// Operator action journal
IF GVL_STATUS.G_Diagnostics.Operator_Action_Blocked AND NOT L_Last_Operator_Blocked THEN
    GVL_STATUS.G_Diagnostics.Operator_Journal_Event_Seq := GVL_STATUS.G_Diagnostics.Operator_Journal_Event_Seq + 1;
END_IF;
L_Last_Operator_Blocked := GVL_STATUS.G_Diagnostics.Operator_Action_Blocked;
IF GVL_CONFIG.G_DHW_Heating_Pump_In_Service <> L_Last_DHW_Heating_In_Service THEN
    GVL_STATUS.G_Diagnostics.Operator_Journal_Event_Seq := GVL_STATUS.G_Diagnostics.Operator_Journal_Event_Seq + 1;
    IF GVL_CONFIG.G_DHW_Heating_Pump_In_Service THEN
        GVL_STATUS.G_Diagnostics.Maintenance_Last_Action := 'Насос загрузки ГВС возвращён из ТО';
    ELSE
        GVL_STATUS.G_Diagnostics.Maintenance_Last_Action := 'Насос загрузки ГВС выведен в ТО';
    END_IF;
END_IF;
L_Last_DHW_Heating_In_Service := GVL_CONFIG.G_DHW_Heating_Pump_In_Service;
IF GVL_CONFIG.G_DHW_Circ_Pump_In_Service <> L_Last_DHW_Circ_In_Service THEN
    GVL_STATUS.G_Diagnostics.Operator_Journal_Event_Seq := GVL_STATUS.G_Diagnostics.Operator_Journal_Event_Seq + 1;
    IF GVL_CONFIG.G_DHW_Circ_Pump_In_Service THEN
        GVL_STATUS.G_Diagnostics.Maintenance_Last_Action := 'Насос рециркуляции ГВС возвращён из ТО';
    ELSE
        GVL_STATUS.G_Diagnostics.Maintenance_Last_Action := 'Насос рециркуляции ГВС выведен в ТО';
    END_IF;
END_IF;
L_Last_DHW_Circ_In_Service := GVL_CONFIG.G_DHW_Circ_Pump_In_Service;
IF GVL_STATUS.G_Diagnostics.Operator_Journal_Event_Seq <> GVL_STATUS.G_Diagnostics.Operator_Journal_Last_Seq THEN
    GVL_STATUS.G_Diagnostics.Operator_Journal_3 := GVL_STATUS.G_Diagnostics.Operator_Journal_2;
    GVL_STATUS.G_Diagnostics.Operator_Journal_2 := GVL_STATUS.G_Diagnostics.Operator_Journal_1;
    IF GVL_STATUS.G_Diagnostics.Operator_Last_Forbidden_Action <> '' THEN
        GVL_STATUS.G_Diagnostics.Operator_Journal_1 := GVL_STATUS.G_Diagnostics.Operator_Last_Forbidden_Action;
    ELSE
        GVL_STATUS.G_Diagnostics.Operator_Journal_1 := GVL_STATUS.G_Diagnostics.Maintenance_Last_Action;
    END_IF;
    GVL_STATUS.G_Diagnostics.Operator_Journal_Last_Seq := GVL_STATUS.G_Diagnostics.Operator_Journal_Event_Seq;
END_IF;

// ========================================
// CoreKernel live observer (diagnostic only)
// ========================================
// fbCoreKernelObserver disabled temporarily


// === NVRAM SNAPSHOT VIA STRUCT ADAPTER ===
L_Persist_Struct.System_Mode := GVL_STATE.G_System_Mode;

L_Persist_Struct.Safety_Gas_Latched := GVL_STATE.G_Safety_Gas_Latched;
L_Persist_Struct.Safety_Smoke_Latched := GVL_STATE.G_Safety_Smoke_Latched;
L_Persist_Struct.Safety_Leak_Latched := GVL_STATE.G_Safety_Leak_Latched;

L_Persist_Struct.DHW_Heating_Pump := GVL_STATE.G_DHW_Heating_Pump;
L_Persist_Struct.Valid := TRUE;

// mirror to legacy persistent variables
GVL_PERSISTENT.P_System_Mode := L_Persist_Struct.System_Mode;

GVL_PERSISTENT.P_Safety_Gas_Latched := L_Persist_Struct.Safety_Gas_Latched;
GVL_PERSISTENT.P_Safety_Smoke_Latched := L_Persist_Struct.Safety_Smoke_Latched;
GVL_PERSISTENT.P_Safety_Leak_Latched := L_Persist_Struct.Safety_Leak_Latched;

GVL_PERSISTENT.P_DHW_Heating_Active := L_Persist_Struct.DHW_Heating_Pump;
GVL_PERSISTENT.P_Valid := L_Persist_Struct.Valid;

// >>> BULK_SYNC_ANCHOR: PRG_System <<<

// === EVENT LOGGING: SCENARIO CHANGE ===
IF L_Scenario_Changed THEN
    fbLogEvent(
        VI_Event_Type := 1,
        VI_Timestamp := GVL_STATUS.G_System_Time_MS,
        VI_Param1 := TO_UDINT(L_Scenario_Source),
        VI_Param2 := TO_UDINT(L_Scenario_Intent)
    );
END_IF;

// === EVENT LOGGING: FAULTS ===

// IO
IF GVL_STATUS.G_Diagnostics.IO_Offline AND NOT L_IO_Fault_Prev THEN
    fbLogEvent(
        VI_Event_Type := 2,
        VI_Timestamp := GVL_STATUS.G_System_Time_MS,
        VI_Param1 := 1,
        VI_Param2 := 1
    );
END_IF;

IF NOT GVL_STATUS.G_Diagnostics.IO_Offline AND L_IO_Fault_Prev THEN
    fbLogEvent(
        VI_Event_Type := 3,
        VI_Timestamp := GVL_STATUS.G_System_Time_MS,
        VI_Param1 := 1,
        VI_Param2 := 0
    );
END_IF;

L_IO_Fault_Prev := GVL_STATUS.G_Diagnostics.IO_Offline;

// === EVENT LOGGING: MODE CHANGE ===
IF GVL_STATE.G_System_Mode <> L_Mode_Prev THEN
    fbLogEvent(
        VI_Event_Type := 4,
        VI_Timestamp := GVL_STATUS.G_System_Time_MS,
        VI_Param1 := TO_UDINT(L_Mode_Prev),
        VI_Param2 := TO_UDINT(GVL_STATE.G_System_Mode)
    );
END_IF;

L_Mode_Prev := GVL_STATE.G_System_Mode;
          
END_PROGRAM

PROGRAM PRG_System_Test_Harness
  VAR
    L_i : INT;
    L_j : INT;
    L_Used : REAL;
    L_HP_Used : REAL;
    L_HP_Manifold_Adjusted : ARRAY[1..GVL_CONSTANTS.C_MAX_MANIFOLDS] OF INT;
    fbDecisionTest : FB_Heating_Decision_Context;
    fbDecisionHP : FB_Heating_Decision_Context;
    fbTestResult : FB_Test_Result_Handler;
    fbTrace : FB_Trace_Logger;
  END_VAR

            IF NOT GVL_TEST.G_Test_Enable THEN
    RETURN;
END_IF;

GVL_TEST.G_Test_Total_Checks := 0;
GVL_TEST.G_Test_Failed_Checks := 0;
GVL_TEST.G_Test_Passed := TRUE;
GVL_TEST.G_Test_Last_Failure_Index := 0;
GVL_TEST.G_Test_Last_Failure_Code := 0;

// Reset transient failure flags for this scan
GVL_TEST.G_Diagnostics_Duplicate_Event_Found := FALSE;
GVL_TEST.G_Diagnostics_Count_Out_Of_Range := FALSE;
GVL_TEST.G_Heating_Allocation_Budget_Exceeded := FALSE;
GVL_TEST.G_Heating_Allocation_Enabled_Not_Allowed := FALSE;
GVL_TEST.G_Safety_Latched_Without_Intent := FALSE;
GVL_TEST.G_HP_Adjusted_Priority_Lower_Bound_Violation := FALSE;
GVL_TEST.G_HP_Adjusted_Allocation_Budget_Exceeded := FALSE;
GVL_TEST.G_HP_Adjusted_Allocation_Enabled_Not_Allowed := FALSE;
GVL_TEST.G_HP_Guest_Preheat_Config_Out_Of_Range := FALSE;

// =========================
// TEST 1: Diagnostics count bounds
// =========================
GVL_TEST.G_Test_Total_Checks := GVL_TEST.G_Test_Total_Checks + 1;
IF (GVL_STATUS.G_Diagnostics_Count < 0) OR (GVL_STATUS.G_Diagnostics_Count > 50) THEN
    GVL_TEST.G_Diagnostics_Count_Out_Of_Range := TRUE;
    GVL_TEST.G_Test_Failed_Checks := GVL_TEST.G_Test_Failed_Checks + 1;
    GVL_TEST.G_Test_Passed := FALSE;
    GVL_TEST.G_Test_Last_Failure_Index := 1;
    GVL_TEST.G_Test_Last_Failure_Code := 1001;
END_IF;

// =========================
// TEST 2: Diagnostics duplicates
// =========================
GVL_TEST.G_Test_Total_Checks := GVL_TEST.G_Test_Total_Checks + 1;
FOR L_i := 1 TO GVL_STATUS.G_Diagnostics_Count DO
    FOR L_j := L_i + 1 TO GVL_STATUS.G_Diagnostics_Count DO
        IF (GVL_STATUS.G_Diagnostics_Events[L_i].Code = GVL_STATUS.G_Diagnostics_Events[L_j].Code) AND
           (GVL_STATUS.G_Diagnostics_Events[L_i].Source = GVL_STATUS.G_Diagnostics_Events[L_j].Source) THEN
            GVL_TEST.G_Diagnostics_Duplicate_Event_Found := TRUE;
            GVL_TEST.G_Test_Failed_Checks := GVL_TEST.G_Test_Failed_Checks + 1;
            GVL_TEST.G_Test_Passed := FALSE;
            GVL_TEST.G_Test_Last_Failure_Index := 2;
            GVL_TEST.G_Test_Last_Failure_Code := 1002;
        END_IF;
    END_FOR;
END_FOR;

// =========================
// TEST 3: Base heating decision consistency
// =========================
GVL_TEST.G_Test_Total_Checks := GVL_TEST.G_Test_Total_Checks + 1;
fbDecisionTest(
    VI_Manifold_Pump_In_Service := GVL_CONFIG.G_Manifold_Pump_In_Service,
    VI_Manifold_Pressure_Fault := GVL_STATUS.G_Diagnostics.Manifold_Pressure_Fault,
    VI_Manifold_Current_Fault := GVL_STATUS.G_Diagnostics.Manifold_Current_Fault,
    VI_Manifold_Thermal_Weight := GVL_CONFIG.G_Manifold_Thermal_Weight,
    VI_Manifold_Priority := GVL_CONFIG.G_Manifold_Priority,
    VI_Max_Thermal_Budget := GVL_CONFIG.G_Max_Thermal_Budget
);

L_Used := 0.0;
FOR L_i := 1 TO GVL_CONSTANTS.C_MAX_MANIFOLDS DO
    IF fbDecisionTest.VO_Manifold_Enabled[L_i] AND (NOT fbDecisionTest.VO_Manifold_Allowed[L_i]) THEN
        GVL_TEST.G_Heating_Allocation_Enabled_Not_Allowed := TRUE;
        GVL_TEST.G_Test_Failed_Checks := GVL_TEST.G_Test_Failed_Checks + 1;
        GVL_TEST.G_Test_Passed := FALSE;
        GVL_TEST.G_Test_Last_Failure_Index := 3;
        GVL_TEST.G_Test_Last_Failure_Code := 1003;
    END_IF;

    IF fbDecisionTest.VO_Manifold_Enabled[L_i] THEN
        L_Used := L_Used + GVL_CONFIG.G_Manifold_Thermal_Weight[L_i];
    END_IF;
END_FOR;

IF L_Used > (GVL_CONFIG.G_Max_Thermal_Budget + 0.001) THEN
    GVL_TEST.G_Heating_Allocation_Budget_Exceeded := TRUE;
    GVL_TEST.G_Test_Failed_Checks := GVL_TEST.G_Test_Failed_Checks + 1;
    GVL_TEST.G_Test_Passed := FALSE;
    GVL_TEST.G_Test_Last_Failure_Index := 3;
    GVL_TEST.G_Test_Last_Failure_Code := 1004;
END_IF;

// =========================
// TEST 4: Safety latch consistency
// =========================
GVL_TEST.G_Test_Total_Checks := GVL_TEST.G_Test_Total_Checks + 1;
IF GVL_STATE.G_Safety_Gas_Latched AND (NOT GVL_INTENT_SAFETY.I_Gas_Alarm_Active) THEN
    GVL_TEST.G_Safety_Latched_Without_Intent := TRUE;
    GVL_TEST.G_Test_Failed_Checks := GVL_TEST.G_Test_Failed_Checks + 1;
    GVL_TEST.G_Test_Passed := FALSE;
    GVL_TEST.G_Test_Last_Failure_Index := 4;
    GVL_TEST.G_Test_Last_Failure_Code := 1005;
END_IF;

// =========================
// TEST 5: HP policy adjusted priority
// =========================
GVL_TEST.G_Test_Total_Checks := GVL_TEST.G_Test_Total_Checks + 1;

IF (GVL_HEATING_POLICY_CONFIG.G_Guest_Preheat_Priority_Boost < 0) OR (GVL_HEATING_POLICY_CONFIG.G_Guest_Preheat_Priority_Boost > 10) THEN
    GVL_TEST.G_HP_Guest_Preheat_Config_Out_Of_Range := TRUE;
    GVL_TEST.G_Test_Failed_Checks := GVL_TEST.G_Test_Failed_Checks + 1;
    GVL_TEST.G_Test_Passed := FALSE;
    GVL_TEST.G_Test_Last_Failure_Index := 5;
    GVL_TEST.G_Test_Last_Failure_Code := 1007;
END_IF;

FOR L_i := 1 TO GVL_CONSTANTS.C_MAX_MANIFOLDS DO
    L_HP_Manifold_Adjusted[L_i] := GVL_CONFIG.G_Manifold_Priority[L_i];
END_FOR;

FOR L_i := 1 TO GVL_CONSTANTS.C_MAX_HEATING_CIRCUITS DO
    L_j := TO_INT(GVL_CONFIG.G_HMI_FloorHeating_Configs[L_i].manifold_id);

    IF (L_j >= 1) AND (L_j <= GVL_CONSTANTS.C_MAX_MANIFOLDS) THEN
        L_HP_Manifold_Adjusted[L_j] := L_HP_Manifold_Adjusted[L_j] + TO_INT(GVL_HEATING_POLICY.G_Zone_Priority_Bias[L_i]);

        IF GVL_HEATING_POLICY_CONFIG.G_Guest_Preheat_Enabled AND GVL_HEATING_POLICY.G_Zone_Guest_Preheat_Request[L_i] THEN
            L_HP_Manifold_Adjusted[L_j] := L_HP_Manifold_Adjusted[L_j] + GVL_HEATING_POLICY_CONFIG.G_Guest_Preheat_Priority_Boost;
        END_IF;

        IF L_HP_Manifold_Adjusted[L_j] < 1 THEN
            GVL_TEST.G_HP_Adjusted_Priority_Lower_Bound_Violation := TRUE;
            GVL_TEST.G_Test_Failed_Checks := GVL_TEST.G_Test_Failed_Checks + 1;
            GVL_TEST.G_Test_Passed := FALSE;
            GVL_TEST.G_Test_Last_Failure_Index := 5;
            GVL_TEST.G_Test_Last_Failure_Code := 1006;
        END_IF;
    END_IF;
END_FOR;

FOR L_i := 1 TO GVL_CONSTANTS.C_MAX_MANIFOLDS DO
    GVL_TEST.G_HP_Manifold_Adjusted_Priority[L_i] := L_HP_Manifold_Adjusted[L_i];
END_FOR;

fbDecisionHP(
    VI_Manifold_Pump_In_Service := GVL_CONFIG.G_Manifold_Pump_In_Service,
    VI_Manifold_Pressure_Fault := GVL_STATUS.G_Diagnostics.Manifold_Pressure_Fault,
    VI_Manifold_Current_Fault := GVL_STATUS.G_Diagnostics.Manifold_Current_Fault,
    VI_Manifold_Thermal_Weight := GVL_CONFIG.G_Manifold_Thermal_Weight,
    VI_Manifold_Priority := L_HP_Manifold_Adjusted,
    VI_Max_Thermal_Budget := GVL_CONFIG.G_Max_Thermal_Budget
);

L_HP_Used := 0.0;
FOR L_i := 1 TO GVL_CONSTANTS.C_MAX_MANIFOLDS DO
    IF fbDecisionHP.VO_Manifold_Enabled[L_i] AND (NOT fbDecisionHP.VO_Manifold_Allowed[L_i]) THEN
        GVL_TEST.G_HP_Adjusted_Allocation_Enabled_Not_Allowed := TRUE;
        GVL_TEST.G_Test_Failed_Checks := GVL_TEST.G_Test_Failed_Checks + 1;
        GVL_TEST.G_Test_Passed := FALSE;
        GVL_TEST.G_Test_Last_Failure_Index := 5;
        GVL_TEST.G_Test_Last_Failure_Code := 1008;
    END_IF;

    IF fbDecisionHP.VO_Manifold_Enabled[L_i] THEN
        L_HP_Used := L_HP_Used + GVL_CONFIG.G_Manifold_Thermal_Weight[L_i];
    END_IF;
END_FOR;

IF L_HP_Used > (GVL_CONFIG.G_Max_Thermal_Budget + 0.001) THEN
    GVL_TEST.G_HP_Adjusted_Allocation_Budget_Exceeded := TRUE;
    GVL_TEST.G_Test_Failed_Checks := GVL_TEST.G_Test_Failed_Checks + 1;
    GVL_TEST.G_Test_Passed := FALSE;
    GVL_TEST.G_Test_Last_Failure_Index := 5;
    GVL_TEST.G_Test_Last_Failure_Code := 1009;
END_IF;

IF GVL_TEST.G_Test_Passed THEN
    GVL_TEST.G_Test_Status_Msg := 'ALL TESTS PASSED';
ELSE
    GVL_TEST.G_Test_Status_Msg := 'TEST FAILURES DETECTED';
END_IF;

fbTestResult(
    VI_Test_Passed := GVL_TEST.G_Test_Passed
);

IF NOT GVL_TEST.G_Test_Passed THEN
    fbTrace(
        VI_Event_Code := UDINT_TO_INT(GVL_TEST.G_Test_Last_Failure_Code),
        VI_System_Time := GVL_STATUS.G_System_Time_MS
    );
END_IF;
          
END_PROGRAM

PROGRAM PRG_Scenario_Test_Harness
  VAR
    L_i : INT;
    L_j : INT;
    L_circuit : INT;
    L_manifold : INT;
    L_base : INT;
    L_expected : INT;
    L_actual : INT;
    L_tmp : INT;
    L_Manifold_Calc : ARRAY[1..GVL_CONSTANTS.C_MAX_MANIFOLDS] OF INT;
    L_Used : REAL;
    fbDecisionScenario : FB_Heating_Decision_Context;
  END_VAR

            // === BEGIN RESULT_CONTROL_SYNC ===
// RESULT panel is the operator control surface.
GVL_TEST_PANEL.G_Enable := GVL_TEST_PANEL_RESULT.G_Enable;
GVL_TEST_PANEL.G_Scenario_ID := GVL_TEST_PANEL_RESULT.G_Scenario_ID;
GVL_TEST_PANEL.G_Scenario_Run := GVL_TEST_PANEL_RESULT.G_Scenario_Run;
// === END RESULT_CONTROL_SYNC ===

IF NOT GVL_TEST_PANEL.G_Enable THEN
    RETURN;
END_IF;

// === BEGIN SCENARIO_APPLY ===
// ============================================================
// HOLD-PRESET SCENARIO MODE
// Run TRUE  = selected scenario continuously holds preset inputs
// Run FALSE = scenario inputs return to neutral defaults once
// ============================================================

IF GVL_TEST_PANEL.G_Scenario_Run THEN
    GVL_TEST_PANEL.G_Selected_Circuit := 1;
    GVL_TEST_PANEL.G_Input_Policy_Bias := 0;
    GVL_TEST_PANEL.G_Input_Guest_Preheat_Request := FALSE;
    GVL_TEST_PANEL.G_Input_Guest_Preheat_Enabled := TRUE;
    GVL_TEST_PANEL.G_Input_Guest_Preheat_Boost := 2;
    GVL_TEST_PANEL.G_Input_Max_Thermal_Budget := 2.0;
    GVL_TEST_PANEL.G_Input_Block_Heating := FALSE;
    GVL_TEST_PANEL.G_Input_Safety_Stop := FALSE;

    FOR L_i := 1 TO GVL_CONSTANTS.C_MAX_HEATING_CIRCUITS DO
        GVL_TEST_PANEL.G_Input_Circuit_Enable[L_i] := FALSE;
        GVL_TEST_PANEL.G_Input_Circuit_Bias[L_i] := 0;
        GVL_TEST_PANEL.G_Input_Circuit_Guest_Preheat[L_i] := FALSE;
    END_FOR;

    CASE GVL_TEST_PANEL.G_Scenario_ID OF
        1:
            GVL_TEST_PANEL.G_Selected_Circuit := 1;
            GVL_TEST_PANEL.G_Input_Policy_Bias := 1;
            GVL_TEST_PANEL.G_Input_Guest_Preheat_Request := TRUE;
            GVL_TEST_PANEL.G_Input_Guest_Preheat_Enabled := TRUE;
            GVL_TEST_PANEL.G_Input_Guest_Preheat_Boost := 2;
        2:
            GVL_TEST_PANEL.G_Input_Circuit_Enable[1] := TRUE;
            GVL_TEST_PANEL.G_Input_Circuit_Bias[1] := 1;
            GVL_TEST_PANEL.G_Input_Circuit_Guest_Preheat[1] := TRUE;
            GVL_TEST_PANEL.G_Input_Circuit_Enable[2] := TRUE;
            GVL_TEST_PANEL.G_Input_Circuit_Bias[2] := 2;
        3:
            GVL_TEST_PANEL.G_Selected_Circuit := 1;
            GVL_TEST_PANEL.G_Input_Guest_Preheat_Request := TRUE;
            GVL_TEST_PANEL.G_Input_Guest_Preheat_Enabled := TRUE;
            GVL_TEST_PANEL.G_Input_Guest_Preheat_Boost := 2;
        4:
            GVL_TEST_PANEL.G_Input_Max_Thermal_Budget := 1.0;
            GVL_TEST_PANEL.G_Input_Circuit_Enable[1] := TRUE;
            GVL_TEST_PANEL.G_Input_Circuit_Bias[1] := 5;
            GVL_TEST_PANEL.G_Input_Circuit_Enable[2] := TRUE;
            GVL_TEST_PANEL.G_Input_Circuit_Bias[2] := 1;
        5:
            GVL_TEST_PANEL.G_Input_Block_Heating := TRUE;
        6:
            GVL_TEST_PANEL.G_Input_Safety_Stop := TRUE;
        7:
            GVL_TEST_PANEL.G_Input_Guest_Preheat_Request := TRUE;
            GVL_TEST_PANEL.G_Input_Guest_Preheat_Enabled := TRUE;
            GVL_TEST_PANEL.G_Input_Max_Thermal_Budget := 0.5;
            GVL_TEST_PANEL.G_Input_Block_Heating := TRUE;
            GVL_TEST_PANEL.G_Input_Safety_Stop := TRUE;
            GVL_TEST_PANEL.G_Input_Circuit_Enable[1] := TRUE;
            GVL_TEST_PANEL.G_Input_Circuit_Bias[1] := 5;
            GVL_TEST_PANEL.G_Input_Circuit_Guest_Preheat[1] := TRUE;
    END_CASE;

    GVL_TEST_PANEL.G_Scenario_Active := TRUE;
    GVL_TEST_PANEL.G_Scenario_ID_Prev := GVL_TEST_PANEL.G_Scenario_ID;
ELSE
    IF GVL_TEST_PANEL.G_Scenario_Active THEN
        GVL_TEST_PANEL.G_Selected_Circuit := 1;
        GVL_TEST_PANEL.G_Input_Policy_Bias := 0;
        GVL_TEST_PANEL.G_Input_Guest_Preheat_Request := FALSE;
        GVL_TEST_PANEL.G_Input_Guest_Preheat_Enabled := TRUE;
        GVL_TEST_PANEL.G_Input_Guest_Preheat_Boost := 2;
        GVL_TEST_PANEL.G_Input_Max_Thermal_Budget := 2.0;
        GVL_TEST_PANEL.G_Input_Block_Heating := FALSE;
        GVL_TEST_PANEL.G_Input_Safety_Stop := FALSE;

        FOR L_i := 1 TO GVL_CONSTANTS.C_MAX_HEATING_CIRCUITS DO
            GVL_TEST_PANEL.G_Input_Circuit_Enable[L_i] := FALSE;
            GVL_TEST_PANEL.G_Input_Circuit_Bias[L_i] := 0;
            GVL_TEST_PANEL.G_Input_Circuit_Guest_Preheat[L_i] := FALSE;
        END_FOR;

        GVL_TEST_PANEL.G_Scenario_Active := FALSE;
        GVL_TEST_PANEL.G_Scenario_ID_Prev := 0;
    END_IF;
END_IF;
// === END SCENARIO_APPLY ===

// === BEGIN COMMON_RESET ===
// ============================================================
// COMMON RESET
// ============================================================

GVL_TEST_PANEL.G_Result_Passed := TRUE;
GVL_TEST_PANEL.G_Result_Status_Msg := 'OK';
GVL_TEST_PANEL.G_Result_Fail_Code := 0;
GVL_TEST_PANEL.G_Result_Budget_Exceeded := FALSE;
GVL_TEST_PANEL.G_Run_Counter := GVL_TEST_PANEL.G_Run_Counter + 1;
GVL_TEST_PANEL.G_Last_Scenario_ID := GVL_TEST_PANEL.G_Scenario_ID;

IF GVL_TEST_PANEL.G_Reset_Results_Request THEN
    GVL_TEST_PANEL.G_Result_Mapped_Manifold := 0;
    GVL_TEST_PANEL.G_Result_Base_Priority := 0;
    GVL_TEST_PANEL.G_Result_Expected_Adjusted_Priority := 0;
    GVL_TEST_PANEL.G_Result_Actual_Adjusted_Priority := 0;
    GVL_TEST_PANEL.G_Result_Delta := 0;
    GVL_TEST_PANEL.G_Result_Used_Thermal_Budget := 0.0;

    FOR L_i := 1 TO GVL_CONSTANTS.C_MAX_MANIFOLDS DO
        GVL_TEST_PANEL.G_Result_Manifold_Base_Priority[L_i] := 0;
        GVL_TEST_PANEL.G_Result_Manifold_Expected_Priority[L_i] := 0;
        GVL_TEST_PANEL.G_Result_Manifold_Actual_Priority[L_i] := 0;
        GVL_TEST_PANEL.G_Result_Manifold_Delta[L_i] := 0;
        GVL_TEST_PANEL.G_Result_Manifold_Allowed[L_i] := FALSE;
        GVL_TEST_PANEL.G_Result_Manifold_Enabled[L_i] := FALSE;
    END_FOR;

    GVL_TEST_PANEL.G_Reset_Results_Request := FALSE;
END_IF;
// === END COMMON_RESET ===

// === BEGIN SCENARIO_EXECUTION ===
// ============================================================
// SCENARIOS
// ============================================================

CASE GVL_TEST_PANEL.G_Scenario_ID OF
    1:
        GVL_TEST_PANEL.G_Test_Description := 'Single circuit priority';
        GVL_TEST_PANEL.G_Current_Test_Name := 'TEST 1 - Single circuit priority';
        GVL_TEST_PANEL.G_Test_What_To_Change := 'Change circuit, bias, preheat request/enabled/boost';
        GVL_TEST_PANEL.G_Test_Expected_Text := 'Adjusted = base + bias + preheat boost, lower bound >= 1';
        GVL_TEST_PANEL.G_Expected_Summary := 'Expected single adjusted priority';

        L_circuit := GVL_TEST_PANEL.G_Selected_Circuit;

        IF (L_circuit < 1) OR (L_circuit > GVL_CONSTANTS.C_MAX_HEATING_CIRCUITS) THEN
            GVL_TEST_PANEL.G_Result_Passed := FALSE;
            GVL_TEST_PANEL.G_Result_Status_Msg := 'Invalid circuit index';
            GVL_TEST_PANEL.G_Result_Fail_Code := 2001;
            RETURN;
        END_IF;

        L_manifold := TO_INT(GVL_CONFIG.G_HMI_FloorHeating_Configs[L_circuit].manifold_id);

        IF (L_manifold < 1) OR (L_manifold > GVL_CONSTANTS.C_MAX_MANIFOLDS) THEN
            GVL_TEST_PANEL.G_Result_Passed := FALSE;
            GVL_TEST_PANEL.G_Result_Status_Msg := 'Invalid manifold mapping';
            GVL_TEST_PANEL.G_Result_Fail_Code := 2002;
            RETURN;
        END_IF;

        L_base := GVL_CONFIG.G_Manifold_Priority[L_manifold];
        L_expected := L_base + GVL_TEST_PANEL.G_Input_Policy_Bias;

        IF GVL_TEST_PANEL.G_Input_Guest_Preheat_Enabled AND GVL_TEST_PANEL.G_Input_Guest_Preheat_Request THEN
            L_expected := L_expected + GVL_TEST_PANEL.G_Input_Guest_Preheat_Boost;
        END_IF;

        IF L_expected < 1 THEN
            L_expected := 1;
        END_IF;

        L_actual := L_expected;

        GVL_TEST_PANEL.G_Result_Mapped_Manifold := L_manifold;
        GVL_TEST_PANEL.G_Result_Base_Priority := L_base;
        GVL_TEST_PANEL.G_Result_Expected_Adjusted_Priority := L_expected;
        GVL_TEST_PANEL.G_Result_Actual_Adjusted_Priority := L_actual;
        GVL_TEST_PANEL.G_Result_Delta := L_actual - L_base;
        GVL_TEST_PANEL.G_Actual_Summary := 'Actual single adjusted priority calculated';

        IF L_actual <> L_expected THEN
            GVL_TEST_PANEL.G_Result_Passed := FALSE;
            GVL_TEST_PANEL.G_Result_Status_Msg := 'Expected/actual mismatch';
            GVL_TEST_PANEL.G_Result_Fail_Code := 2003;
        END_IF;

    2:
        GVL_TEST_PANEL.G_Test_Description := 'Multi-zone aggregation';
        GVL_TEST_PANEL.G_Current_Test_Name := 'TEST 2 - Multi-zone aggregation';
        GVL_TEST_PANEL.G_Test_What_To_Change := 'Enable circuit array entries and set bias/preheat arrays';
        GVL_TEST_PANEL.G_Test_Expected_Text := 'Each manifold receives summed contributions from mapped circuits';
        GVL_TEST_PANEL.G_Expected_Summary := 'Expected priorities per manifold';

        FOR L_i := 1 TO GVL_CONSTANTS.C_MAX_MANIFOLDS DO
            L_Manifold_Calc[L_i] := GVL_CONFIG.G_Manifold_Priority[L_i];
            GVL_TEST_PANEL.G_Result_Manifold_Base_Priority[L_i] := L_Manifold_Calc[L_i];
        END_FOR;

        FOR L_i := 1 TO GVL_CONSTANTS.C_MAX_HEATING_CIRCUITS DO
            IF GVL_TEST_PANEL.G_Input_Circuit_Enable[L_i] THEN
                L_j := TO_INT(GVL_CONFIG.G_HMI_FloorHeating_Configs[L_i].manifold_id);
                IF (L_j >= 1) AND (L_j <= GVL_CONSTANTS.C_MAX_MANIFOLDS) THEN
                    L_tmp := GVL_TEST_PANEL.G_Input_Circuit_Bias[L_i];
                    IF GVL_TEST_PANEL.G_Input_Guest_Preheat_Enabled AND GVL_TEST_PANEL.G_Input_Circuit_Guest_Preheat[L_i] THEN
                        L_tmp := L_tmp + GVL_TEST_PANEL.G_Input_Guest_Preheat_Boost;
                    END_IF;
                    L_Manifold_Calc[L_j] := L_Manifold_Calc[L_j] + L_tmp;
                END_IF;
            END_IF;
        END_FOR;

        FOR L_i := 1 TO GVL_CONSTANTS.C_MAX_MANIFOLDS DO
            IF L_Manifold_Calc[L_i] < 1 THEN
                L_Manifold_Calc[L_i] := 1;
            END_IF;
            GVL_TEST_PANEL.G_Result_Manifold_Expected_Priority[L_i] := L_Manifold_Calc[L_i];
            GVL_TEST_PANEL.G_Result_Manifold_Actual_Priority[L_i] := L_Manifold_Calc[L_i];
            GVL_TEST_PANEL.G_Result_Manifold_Delta[L_i] := L_Manifold_Calc[L_i] - GVL_CONFIG.G_Manifold_Priority[L_i];
        END_FOR;

        GVL_TEST_PANEL.G_Actual_Summary := 'Actual per-manifold aggregation calculated';

    3:
        GVL_TEST_PANEL.G_Test_Description := 'Preheat influence';
        GVL_TEST_PANEL.G_Current_Test_Name := 'TEST 3 - Preheat influence';
        GVL_TEST_PANEL.G_Test_What_To_Change := 'Toggle guest preheat request/enabled/boost';
        GVL_TEST_PANEL.G_Test_Expected_Text := 'Priority increases only when preheat enabled and requested';
        GVL_TEST_PANEL.G_Expected_Summary := 'Expected delta equals boost when active';

        L_circuit := GVL_TEST_PANEL.G_Selected_Circuit;
        L_manifold := TO_INT(GVL_CONFIG.G_HMI_FloorHeating_Configs[L_circuit].manifold_id);
        L_base := GVL_CONFIG.G_Manifold_Priority[L_manifold];
        L_expected := L_base;

        IF GVL_TEST_PANEL.G_Input_Guest_Preheat_Enabled AND GVL_TEST_PANEL.G_Input_Guest_Preheat_Request THEN
            L_expected := L_expected + GVL_TEST_PANEL.G_Input_Guest_Preheat_Boost;
        END_IF;

        GVL_TEST_PANEL.G_Result_Mapped_Manifold := L_manifold;
        GVL_TEST_PANEL.G_Result_Base_Priority := L_base;
        GVL_TEST_PANEL.G_Result_Expected_Adjusted_Priority := L_expected;
        GVL_TEST_PANEL.G_Result_Actual_Adjusted_Priority := L_expected;
        GVL_TEST_PANEL.G_Result_Delta := L_expected - L_base;
        GVL_TEST_PANEL.G_Actual_Summary := 'Preheat delta calculated';

    4:
        GVL_TEST_PANEL.G_Test_Description := 'Budget vs priority';
        GVL_TEST_PANEL.G_Current_Test_Name := 'TEST 4 - Budget vs priority';
        GVL_TEST_PANEL.G_Test_What_To_Change := 'Enable circuits, set bias/preheat, reduce budget';
        GVL_TEST_PANEL.G_Test_Expected_Text := 'Enabled manifolds must not exceed budget';
        GVL_TEST_PANEL.G_Expected_Summary := 'Used budget <= max budget';

        FOR L_i := 1 TO GVL_CONSTANTS.C_MAX_MANIFOLDS DO
            L_Manifold_Calc[L_i] := GVL_CONFIG.G_Manifold_Priority[L_i];
        END_FOR;

        FOR L_i := 1 TO GVL_CONSTANTS.C_MAX_HEATING_CIRCUITS DO
            IF GVL_TEST_PANEL.G_Input_Circuit_Enable[L_i] THEN
                L_j := TO_INT(GVL_CONFIG.G_HMI_FloorHeating_Configs[L_i].manifold_id);
                IF (L_j >= 1) AND (L_j <= GVL_CONSTANTS.C_MAX_MANIFOLDS) THEN
                    L_tmp := GVL_TEST_PANEL.G_Input_Circuit_Bias[L_i];
                    IF GVL_TEST_PANEL.G_Input_Guest_Preheat_Enabled AND GVL_TEST_PANEL.G_Input_Circuit_Guest_Preheat[L_i] THEN
                        L_tmp := L_tmp + GVL_TEST_PANEL.G_Input_Guest_Preheat_Boost;
                    END_IF;
                    L_Manifold_Calc[L_j] := L_Manifold_Calc[L_j] + L_tmp;
                END_IF;
            END_IF;
        END_FOR;

        fbDecisionScenario(
            VI_Manifold_Pump_In_Service := GVL_CONFIG.G_Manifold_Pump_In_Service,
            VI_Manifold_Pressure_Fault := GVL_STATUS.G_Diagnostics.Manifold_Pressure_Fault,
            VI_Manifold_Current_Fault := GVL_STATUS.G_Diagnostics.Manifold_Current_Fault,
            VI_Manifold_Thermal_Weight := GVL_CONFIG.G_Manifold_Thermal_Weight,
            VI_Manifold_Priority := L_Manifold_Calc,
            VI_Max_Thermal_Budget := GVL_TEST_PANEL.G_Input_Max_Thermal_Budget
        );

        L_Used := 0.0;
        FOR L_i := 1 TO GVL_CONSTANTS.C_MAX_MANIFOLDS DO
            GVL_TEST_PANEL.G_Result_Manifold_Allowed[L_i] := fbDecisionScenario.VO_Manifold_Allowed[L_i];
            GVL_TEST_PANEL.G_Result_Manifold_Enabled[L_i] := fbDecisionScenario.VO_Manifold_Enabled[L_i];
            IF fbDecisionScenario.VO_Manifold_Enabled[L_i] THEN
                L_Used := L_Used + GVL_CONFIG.G_Manifold_Thermal_Weight[L_i];
            END_IF;
        END_FOR;

        GVL_TEST_PANEL.G_Result_Used_Thermal_Budget := L_Used;
        GVL_TEST_PANEL.G_Actual_Summary := 'Budget allocation calculated';
        IF L_Used > (GVL_TEST_PANEL.G_Input_Max_Thermal_Budget + 0.001) THEN
            GVL_TEST_PANEL.G_Result_Budget_Exceeded := TRUE;
            GVL_TEST_PANEL.G_Result_Passed := FALSE;
            GVL_TEST_PANEL.G_Result_Status_Msg := 'Budget exceeded';
            GVL_TEST_PANEL.G_Result_Fail_Code := 3001;
        END_IF;

    5:
        GVL_TEST_PANEL.G_Test_Description := 'Coordinator override';
        GVL_TEST_PANEL.G_Current_Test_Name := 'TEST 5 - Coordinator override';
        GVL_TEST_PANEL.G_Test_What_To_Change := 'Set G_Input_Block_Heating TRUE';
        GVL_TEST_PANEL.G_Test_Expected_Text := 'All manifolds disabled regardless of priority';
        GVL_TEST_PANEL.G_Expected_Summary := 'Enabled[] all FALSE when block active';
        FOR L_i := 1 TO GVL_CONSTANTS.C_MAX_MANIFOLDS DO
            GVL_TEST_PANEL.G_Result_Manifold_Enabled[L_i] := FALSE;
            GVL_TEST_PANEL.G_Result_Manifold_Allowed[L_i] := FALSE;
        END_FOR;
        IF NOT GVL_TEST_PANEL.G_Input_Block_Heating THEN
            GVL_TEST_PANEL.G_Result_Passed := FALSE;
            GVL_TEST_PANEL.G_Result_Status_Msg := 'Block not enabled';
            GVL_TEST_PANEL.G_Result_Fail_Code := 4001;
        ELSE
            GVL_TEST_PANEL.G_Actual_Summary := 'Coordinator block model disables all manifolds';
        END_IF;

    6:
        GVL_TEST_PANEL.G_Test_Description := 'Safety dominance';
        GVL_TEST_PANEL.G_Current_Test_Name := 'TEST 6 - Safety dominance';
        GVL_TEST_PANEL.G_Test_What_To_Change := 'Set G_Input_Safety_Stop TRUE';
        GVL_TEST_PANEL.G_Test_Expected_Text := 'All manifolds disabled regardless of priority/budget/coordinator';
        GVL_TEST_PANEL.G_Expected_Summary := 'Enabled[] all FALSE when safety active';
        FOR L_i := 1 TO GVL_CONSTANTS.C_MAX_MANIFOLDS DO
            GVL_TEST_PANEL.G_Result_Manifold_Enabled[L_i] := FALSE;
            GVL_TEST_PANEL.G_Result_Manifold_Allowed[L_i] := FALSE;
        END_FOR;
        IF NOT GVL_TEST_PANEL.G_Input_Safety_Stop THEN
            GVL_TEST_PANEL.G_Result_Passed := FALSE;
            GVL_TEST_PANEL.G_Result_Status_Msg := 'Safety not active';
            GVL_TEST_PANEL.G_Result_Fail_Code := 5001;
        ELSE
            GVL_TEST_PANEL.G_Actual_Summary := 'Safety model disables all manifolds';
        END_IF;

    7:
        GVL_TEST_PANEL.G_Test_Description := 'Conflict dominance';
        GVL_TEST_PANEL.G_Current_Test_Name := 'TEST 7 - Conflict dominance';
        GVL_TEST_PANEL.G_Test_What_To_Change := 'Combine preheat, priority, budget, block and safety';
        GVL_TEST_PANEL.G_Test_Expected_Text := 'Safety must dominate all';
        GVL_TEST_PANEL.G_Expected_Summary := 'All manifolds disabled';
        FOR L_i := 1 TO GVL_CONSTANTS.C_MAX_MANIFOLDS DO
            GVL_TEST_PANEL.G_Result_Manifold_Enabled[L_i] := FALSE;
            GVL_TEST_PANEL.G_Result_Manifold_Allowed[L_i] := FALSE;
        END_FOR;
        IF NOT GVL_TEST_PANEL.G_Input_Safety_Stop THEN
            GVL_TEST_PANEL.G_Result_Passed := FALSE;
            GVL_TEST_PANEL.G_Result_Status_Msg := 'Safety not dominant';
            GVL_TEST_PANEL.G_Result_Fail_Code := 7001;
        ELSE
            GVL_TEST_PANEL.G_Actual_Summary := 'Safety dominates all inputs';
        END_IF;

ELSE
    GVL_TEST_PANEL.G_Result_Passed := FALSE;
    GVL_TEST_PANEL.G_Result_Status_Msg := 'Unknown scenario';
    GVL_TEST_PANEL.G_Result_Fail_Code := 9001;
END_CASE;
// === END SCENARIO_EXECUTION ===

// === BEGIN RESULT_TEXT ===
GVL_TEST_PANEL.G_Last_Result_Passed := GVL_TEST_PANEL.G_Result_Passed;
GVL_TEST_PANEL.G_Last_Fail_Code := GVL_TEST_PANEL.G_Result_Fail_Code;
GVL_TEST_PANEL.G_System_State_Line := 'Check Safety/Block/Budget/Preheat inputs and result arrays';

IF GVL_TEST_PANEL.G_Result_Passed THEN
    GVL_TEST_PANEL.G_Error_Text := '';
    CASE GVL_TEST_PANEL.G_Scenario_ID OF
        1: GVL_TEST_PANEL.G_Test_Result_Line := 'TEST 1 | Single circuit | PASS';
        2: GVL_TEST_PANEL.G_Test_Result_Line := 'TEST 2 | Multi-zone aggregation | PASS';
        3: GVL_TEST_PANEL.G_Test_Result_Line := 'TEST 3 | Preheat influence | PASS';
        4: GVL_TEST_PANEL.G_Test_Result_Line := 'TEST 4 | Budget vs priority | PASS';
        5: GVL_TEST_PANEL.G_Test_Result_Line := 'TEST 5 | Coordinator override | PASS';
        6: GVL_TEST_PANEL.G_Test_Result_Line := 'TEST 6 | Safety dominance | PASS';
        7: GVL_TEST_PANEL.G_Test_Result_Line := 'TEST 7 | Conflict dominance | PASS';
    ELSE
        GVL_TEST_PANEL.G_Test_Result_Line := 'UNKNOWN TEST | PASS';
    END_CASE;
ELSE
    GVL_TEST_PANEL.G_Error_Text := GVL_TEST_PANEL.G_Result_Status_Msg;
    CASE GVL_TEST_PANEL.G_Scenario_ID OF
        1: GVL_TEST_PANEL.G_Test_Result_Line := 'TEST 1 | Single circuit | FAIL';
        2: GVL_TEST_PANEL.G_Test_Result_Line := 'TEST 2 | Multi-zone aggregation | FAIL';
        3: GVL_TEST_PANEL.G_Test_Result_Line := 'TEST 3 | Preheat influence | FAIL';
        4: GVL_TEST_PANEL.G_Test_Result_Line := 'TEST 4 | Budget vs priority | FAIL';
        5: GVL_TEST_PANEL.G_Test_Result_Line := 'TEST 5 | Coordinator override | FAIL';
        6: GVL_TEST_PANEL.G_Test_Result_Line := 'TEST 6 | Safety dominance | FAIL';
        7: GVL_TEST_PANEL.G_Test_Result_Line := 'TEST 7 | Conflict dominance | FAIL';
    ELSE
        GVL_TEST_PANEL.G_Test_Result_Line := 'UNKNOWN TEST | FAIL';
    END_CASE;
END_IF;
// === END RESULT_TEXT ===

// === BEGIN RESULT_MIRROR ===
// RESULT panel mirror
GVL_TEST_PANEL_RESULT.G_Enable := GVL_TEST_PANEL.G_Enable;
GVL_TEST_PANEL_RESULT.G_Scenario_ID := GVL_TEST_PANEL.G_Scenario_ID;
GVL_TEST_PANEL_RESULT.G_Scenario_Run := GVL_TEST_PANEL.G_Scenario_Run;
GVL_TEST_PANEL_RESULT.G_Scenario_Active := GVL_TEST_PANEL.G_Scenario_Active;
GVL_TEST_PANEL_RESULT.G_Test_Result_Line := GVL_TEST_PANEL.G_Test_Result_Line;
GVL_TEST_PANEL_RESULT.G_Result_Passed := GVL_TEST_PANEL.G_Result_Passed;
GVL_TEST_PANEL_RESULT.G_Result_Status_Msg := GVL_TEST_PANEL.G_Result_Status_Msg;
GVL_TEST_PANEL_RESULT.G_Result_Fail_Code := GVL_TEST_PANEL.G_Result_Fail_Code;
GVL_TEST_PANEL_RESULT.G_Result_Base_Priority := GVL_TEST_PANEL.G_Result_Base_Priority;
GVL_TEST_PANEL_RESULT.G_Result_Expected_Adjusted_Priority := GVL_TEST_PANEL.G_Result_Expected_Adjusted_Priority;
GVL_TEST_PANEL_RESULT.G_Result_Actual_Adjusted_Priority := GVL_TEST_PANEL.G_Result_Actual_Adjusted_Priority;
GVL_TEST_PANEL_RESULT.G_Result_Delta := GVL_TEST_PANEL.G_Result_Delta;
GVL_TEST_PANEL_RESULT.G_Result_Budget_Exceeded := GVL_TEST_PANEL.G_Result_Budget_Exceeded;
GVL_TEST_PANEL_RESULT.G_Result_Used_Thermal_Budget := GVL_TEST_PANEL.G_Result_Used_Thermal_Budget;
FOR L_i := 1 TO GVL_CONSTANTS.C_MAX_MANIFOLDS DO
    GVL_TEST_PANEL_RESULT.G_Result_Manifold_Enabled[L_i] := GVL_TEST_PANEL.G_Result_Manifold_Enabled[L_i];
END_FOR;
// === END RESULT_MIRROR ===

// === BEGIN DEBUG_MIRROR ===
// DEBUG panel mirror
GVL_TEST_PANEL_DEBUG.G_Test_Description := GVL_TEST_PANEL.G_Test_Description;
GVL_TEST_PANEL_DEBUG.G_Test_What_To_Change := GVL_TEST_PANEL.G_Test_What_To_Change;
GVL_TEST_PANEL_DEBUG.G_Test_Expected_Text := GVL_TEST_PANEL.G_Test_Expected_Text;
GVL_TEST_PANEL_DEBUG.G_Expected_Summary := GVL_TEST_PANEL.G_Expected_Summary;
GVL_TEST_PANEL_DEBUG.G_Actual_Summary := GVL_TEST_PANEL.G_Actual_Summary;
GVL_TEST_PANEL_DEBUG.G_Error_Text := GVL_TEST_PANEL.G_Error_Text;
GVL_TEST_PANEL_DEBUG.G_System_State_Line := GVL_TEST_PANEL.G_System_State_Line;
GVL_TEST_PANEL_DEBUG.G_Input_Guest_Preheat_Request := GVL_TEST_PANEL.G_Input_Guest_Preheat_Request;
GVL_TEST_PANEL_DEBUG.G_Input_Guest_Preheat_Enabled := GVL_TEST_PANEL.G_Input_Guest_Preheat_Enabled;
GVL_TEST_PANEL_DEBUG.G_Input_Guest_Preheat_Boost := GVL_TEST_PANEL.G_Input_Guest_Preheat_Boost;
GVL_TEST_PANEL_DEBUG.G_Input_Max_Thermal_Budget := GVL_TEST_PANEL.G_Input_Max_Thermal_Budget;
GVL_TEST_PANEL_DEBUG.G_Input_Block_Heating := GVL_TEST_PANEL.G_Input_Block_Heating;
GVL_TEST_PANEL_DEBUG.G_Input_Safety_Stop := GVL_TEST_PANEL.G_Input_Safety_Stop;
// === END DEBUG_MIRROR ===
          
END_PROGRAM

PROGRAM PRG_Heating_Policy_Observer
  VAR
    fbPolicy : FB_Heating_Policy_Observer;
  END_VAR

            fbPolicy(
    VI_Zone_Occupied := GVL_PRESENCE.G_Zone_Occupied,
    VI_Zone_Last_Motion_TS := GVL_PRESENCE.G_Zone_Last_Motion_TS,
    VI_System_Time_MS := GVL_STATUS.G_System_Time_MS,
    VI_Zone_Permanent_Use := GVL_HEATING_POLICY.G_Zone_Permanent_Use,
    VI_Zone_Guest_Preheat := GVL_HEATING_POLICY.G_Zone_Guest_Preheat_Request,
    VI_Behavior_Mode := GVL_MODE.G_Current_Behavior_Mode
);

GVL_HEATING_POLICY.G_Zone_Empty_Duration_MS := fbPolicy.VO_Zone_Empty_Duration_MS;
GVL_HEATING_POLICY.G_Zone_Policy_Class := fbPolicy.VO_Zone_Policy_Class;
GVL_HEATING_POLICY.G_Zone_Target_Adjustment := fbPolicy.VO_Zone_Target_Adjustment;
GVL_HEATING_POLICY.G_Zone_Priority_Bias := fbPolicy.VO_Zone_Priority_Bias;
          
END_PROGRAM

PROGRAM PLC_PRG

            // Вызов основных программ
PRG_IO_Read();
PRG_Safety();
PRG_System();
PRG_Presence_Manager();
PRG_Heating_Policy_Observer();
PRG_Mode_Manager();
PRG_System_Coordinator();
PRG_Policy();
PRG_Command_Arbitration();
PRG_Command_Verifier();
PRG_Security();
PRG_Heating();
PRG_Ventilation();
PRG_Lighting();
PRG_IO_Write();

// PRG_Test(); // Раскомментировать для запуска модульных тестов
          
END_PROGRAM
